TEXTLIST visuTextLinks
  A = 'GVL.axes[1].Axis.NcToPlc.ActPos'
   = ''
END_TEXTLIST

(* stored: Version 1.1.0.1, ProductVersion 3.1.4024.5
   TextList visuTextLinks: Id {f7469b03-da64-4a47-8ac8-39435c36424f} *)
